// TIA Portal V18 export
TYPE "LGasp_typeQuota"
// stored: IsFailsafeCompliant false
   STRUCT
      quotax : LReal := -1.0;   // [mm] - posizione asse X
      quotay : LReal := -1.0;   // [mm] - posizione asse Y
      rifcor_y : Int;   // riferimento al correttore della DB L1_Corr_plotter
      quotaz : LReal := -1.0;   // [mm] - posizione asse Z
      gradi : LReal := -1.0;   // [°] - posizione rotazione
      mouldea : Array[1..16] of Bool;   // Punzoni A
      mouldeb : Array[1..16] of Bool;   // Punzoni B
      mouldec : Array[1..16] of Bool;   // Punzoni C
      moulded : Array[1..16] of Bool;   // Punzoni D
      moulde_pos : Array[1..16] of LReal;
      state : Struct
         ultimaquotapezzo : Bool;   // Ultima quota del pezzo
         quotavalida : Bool;   // Quota valida da PC
         quotataglio : Bool;   // Taglio del pezzo T su articolo
         quotatagliocoda : Bool;   // Taglio del pezzo TC su articolo
         quotatagliotesta : Bool;   // Taglio della testa TT su articolo
         bool_5 : Bool;
         bool_6 : Bool;
         bool_7 : Bool;
         bool_8 : Bool;
         bool_9 : Bool;
         bool_10 : Bool;
         bool_11 : Bool;
         bool_12 : Bool;
         bool_13 : Bool;
         bool_14 : Bool;
         bool_15 : Bool;
         bool_16 : Bool;
         bool_17 : Bool;
         bool_18 : Bool;
         bool_19 : Bool;
         bool_20 : Bool;
         bool_21 : Bool;
         bool_22 : Bool;
         bool_23 : Bool;
         bool_24 : Bool;
         bool_25 : Bool;
         bool_26 : Bool;
         bool_27 : Bool;
         bool_28 : Bool;
         bool_29 : Bool;
         bool_30 : Bool;
         bool_31 : Bool;
      END_STRUCT;
      infinitystep : Bool;   // Abilita passo infinito
      print : "LGasp_typeStampante";   // Stampante
   END_STRUCT;
END_TYPE
